// TIA Portal V17 export
// export: Created 2021-09-08T12:46:16.1780561Z, ExportSetting WithDefaults, DisplayName Totally Integrated Automation Portal, DisplayVersion V17, DisplayName TIA Portal Openness, DisplayVersion V17, DisplayName TIA Portal Version Control Interface, DisplayVersion V17, DisplayName STEP 7 Professional, DisplayVersion V17, DisplayName STEP 7 Safety, DisplayVersion V17, DisplayName WinCC Advanced, DisplayVersion V17
DATA_BLOCK "dbVolumeCounters"   // DB10
{ S7_Optimized_Access := 'FALSE' }
VERSION : 1.1
// stored: AutoNumber true, DBAccessibleFromOPCUA true, IsOnlyStoredInLoadMemory false, IsWriteProtectedInAS false
   VAR RETAIN
      FM201 : FREQ_COUNTER;   // Inlet water consumption FM201
      FM501 : FREQ_COUNTER;   // Inlet water consumption UF FM501
      FM502 : FREQ_COUNTER;   // Inlet water consumption UF FM502
      FM901 : FREQ_COUNTER;   // Consumption of permeate RO FM901
      FM902 : FREQ_COUNTER;   // Concentrate consumption RO FM902
      FM1201 : FREQ_COUNTER;   // Consumption of permeate per consumer FM1201
      FM1301 : FREQ_COUNTER;   // Consumption of permeate NF FM1301
      FM1302 : FREQ_COUNTER;   // Concentrate consumption NF FM1302
      FM1701 : FREQ_COUNTER;   // Consumption of nanofiltrate on the consumer FM1701
      FM1801 : FREQ_COUNTER;   // Sewage consumption FM1801
   END_VAR
BEGIN
END_DATA_BLOCK
